# EPICS substitutions: evrSupport/Db/ioc/IOC-IN20-PM05pattern.substitutions
#
# Pattern records
file evrPatternAll.db {
#	    Device        ,  SLC Pattern Check LNK    , EVR/Trigger
#	                                                  Links
  pattern { DEVICE        ,        LINK4              , LINK5 , LINK6 }
	  { IOC:IN20:PM05 ,         ""                ,  ""   ,  ""   }
}
file evrEventAll.db {
  pattern { DEVICE }
	  { IOC:IN20:PM05}
}
